TYPE ST_CapacitorSchemaColorWithDisconnector EXTENDS ST_CapacitorSchemaColorBase :
STRUCT
	DisconnectorPosition : E_DisconnectorPosition;
END_STRUCT
END_TYPE

(* stored: Version 1.1.0.1, ProductVersion 3.1.4024.13
   DUT ST_CapacitorSchemaColorWithDisconnector: Id {9d300a5e-461f-40b4-95bd-a0d4717808f0} *)
